{attribute 'GeneratedUsingTerminal: EL3681-0000-0018'}
{attribute addProperty BoxType "EL3681-0000-0018"}
{attribute addProperty Id "Disable_autorangeBOOL1Start_calibrationBOOL1ModeBYTE1RangeSINT1"}
{attribute addProperty CRC "416629465"}
{attribute addProperty Size "4"}
TYPE Control_18D542D9 :
STRUCT
	{attribute addProperty Name "Disable_autorange"}
	Disable_autorange : BOOL;
	{attribute addProperty Name "Start_calibration"}
	Start_calibration : BOOL;
	{attribute addProperty Name "Mode"}
	Mode : BYTE;
	{attribute addProperty Name "Range"}
	Range : SINT;
END_STRUCT
END_TYPE

(* stored: Version 1.2.0.0, ProductVersion 3.1.4024.11
   DUT Control_18D542D9: Id {43e6354f-4194-43d9-b6a1-1256cd2379a4} *)
